KUKA KRL program: SIGN.src

&ACCESS RV
&REL 1
&PARAM TEMPLATE = C:\KRC\Roboter\Template\FunctionVorgabe
&PARAM EDITMASK = *
DEFFCT REAL SIGN(VALUE:IN )
  REAL VALUE
  REAL RET_VAL
  IF VALUE >= 0.0 THEN
    RET_VAL = 1.0
  ELSE
    RET_VAL = -1.0
  ENDIF

  RETURN(RET_VAL)
ENDFCT
